FUNCTION RUN : BOOL

GVL.fbTcUnitRunner.RunFunctionBlocksTests();

END_FUNCTION

(* stored: Version 1.1.0.1, ProductVersion 3.1.4022.12
   POU RUN: Id {bd49b256-e7ba-4b73-b669-380d1f428417}, SpecialFunc None *)
